Yaskawa INFORM job: X2_34(P)(-165,-90).JBI

/JOB
//NAME X2_34(P)(-165,-90)
//POS
///NPOS 175,175,175,10,0,0
///TOOL 0
///POSTYPE PULSE
///PULSE
C00000=39612,-76551,-106625,-19964,71626,-76894
C00001=136747,-74177,-105509,-19364,71994,-77223
C00002=161484,-91945,-110261,-14957,103238,-71453
C00003=108557,-106327,-63424,-3944,69973,-81240
C00004=108101,-105157,-58666,-3986,67629,-81319
C00005=107910,-104606,-56713,-4004,66704,-81354
C00006=107850,-103240,-54402,-4023,65983,-81349
C00007=107869,-103453,-54807,-4020,66123,-81348
C00008=107897,-103507,-54813,-4022,66100,-81337
C00009=107488,-105602,-55530,-4025,65447,-81456
C00010=107897,-103507,-54813,-4022,66100,-81337
C00011=108089,-104086,-56785,-4002,67023,-81302
C00012=108547,-105331,-61592,-3959,69358,-81223
C00013=104324,-140520,-91585,-2551,64945,-84379
C00014=108507,-122565,-87623,-3050,71648,-81402
C00015=108151,-121446,-83013,-3052,69376,-81469
C00016=108261,-118225,-79182,-3077,68679,-81414
C00017=108248,-117713,-78438,-3081,68485,-81412
C00018=107960,-119858,-79317,-3061,67913,-81499
C00019=108018,-119853,-79323,-3067,67922,-81479
C00020=107613,-122457,-80135,-3040,67069,-81600
C00021=108018,-119853,-79323,-3067,67922,-81479
C00022=108166,-120422,-81226,-3065,68804,-81449
C00023=108523,-121621,-85875,-3062,71060,-81382
C00024=103983,-152784,-104117,29,47198,-80645
C00025=107925,-135086,-100462,-1830,53864,-79007
C00026=108009,-130425,-94870,-1890,52821,-78954
C00027=108095,-127409,-91509,-1942,52305,-78908
C00028=108095,-126631,-90337,-1950,51984,-78902
C00029=107997,-127624,-90886,-1911,51808,-78940
C00030=108092,-127668,-90899,-1953,51796,-78900
C00031=107688,-130656,-91794,-1800,50803,-79052
C00032=108092,-127668,-90899,-1953,51796,-78900
C00033=108059,-129495,-93147,-1927,52240,-78922
C00034=107976,-134157,-98754,-1865,53292,-78976
C00035=177778,-171467,-115875,-22983,53224,-57909
C00036=173225,-131569,-103985,-1828,82945,-64027
C00037=174834,-131579,-99933,-1874,80485,-63443
C00038=175501,-131430,-98256,-1893,79546,-63202
C00039=175652,-130307,-96214,-1900,78870,-63140
C00040=175501,-131430,-98256,-1893,79546,-63202
C00041=175673,-130387,-96489,-1900,78999,-63135
C00042=177249,-132864,-97254,-1939,78235,-62586
C00043=175673,-130387,-96489,-1900,78999,-63135
C00044=175002,-130579,-98183,-1880,79926,-63378
C00045=173387,-130693,-102281,-1834,82351,-63963
C00046=183807,-145514,-102399,-23160,59516,-56806
C00047=173742,-122117,-87314,-5245,73809,-63439
C00048=174955,-120554,-82580,-5392,71786,-62928
C00049=175454,-119846,-80647,-5453,70997,-62718
C00050=175604,-118612,-78506,-5486,70327,-62635
C00051=175579,-118770,-78792,-5481,70420,-62648
C00052=175582,-118807,-78841,-5481,70431,-62647
C00053=177158,-120803,-79498,-5617,69918,-62073
C00054=175582,-118807,-78841,-5481,70431,-62647
C00055=175081,-119542,-80788,-5418,71215,-62858
C00056=173863,-121178,-85561,-5269,73223,-63371
C00057=178906,-130545,-89223,-5416,71014,-61548
C00058=173071,-106231,-63228,-1896,70899,-63899
C00059=174678,-104574,-58322,-1958,68769,-63315
C00060=175345,-103832,-56313,-1985,67930,-63072
C00061=175495,-102440,-53993,-1998,67222,-63009
C00062=175462,-102665,-54381,-1995,67344,-63022
C00063=175499,-102701,-54366,-1997,67317,-63009
C00064=177075,-104318,-54954,-2039,66885,-62461
C00065=175499,-102701,-54366,-1997,67317,-63009
C00066=174829,-103469,-56394,-1970,68154,-63253
C00067=173213,-105197,-61348,-1906,70277,-63841
C00068=156325,-82511,-105508,-20476,72304,-69745
C00069=137289,-84891,-120500,-10173,76813,-76449
C00070=137303,-139323,-128947,-10263,31295,-76421
C00071=31263,-162610,-128854,-9653,11963,-76756
C00072=-11604,-169116,-125244,-11553,23484,-75880
C00073=-126218,-114256,-117174,-36511,17097,-65041
C00074=-135014,-119633,-103449,-15272,86576,-49606
C00075=-106915,-105368,-62725,-601,70273,-77124
C00076=-106469,-104199,-57962,-625,67946,-76958
C00077=-106427,-102978,-55809,-630,67247,-76940
C00078=-106243,-102289,-53695,-641,66303,-76872
C00079=-106247,-102493,-54033,-640,66406,-76874
C00080=-106414,-102537,-54077,-634,66410,-76931
C00081=-105966,-104617,-54795,-653,65787,-76773
C00082=-106414,-102537,-54077,-634,66410,-76931
C00083=-106600,-103115,-56051,-624,67326,-77000
C00084=-107042,-104359,-60863,-599,69645,-77164
C00085=-104685,-138629,-91180,-1583,66049,-76219
C00086=-106630,-121517,-86856,-1571,71994,-76952
C00087=-106291,-120404,-82245,-1626,69736,-76803
C00088=-106369,-118603,-80003,-1623,69281,-76825
C00089=-106273,-117758,-77970,-1641,68465,-76779
C00090=-106369,-117325,-78035,-1630,68726,-76817
C00091=-105806,-121493,-79397,-1702,67435,-76600
C00092=-106260,-118916,-78588,-1645,68251,-76772
C00093=-106400,-119484,-80492,-1621,69128,-76833
C00094=-106737,-120682,-85145,-1565,71368,-76981
C00095=-103582,-154725,-104423,-7901,46985,-74327
C00096=-105847,-133932,-99601,-6432,54310,-75790
C00097=-106008,-129334,-94017,-6450,53230,-75789
C00098=-106186,-126781,-91574,-6391,53025,-75850
C00099=-106032,-126404,-89711,-6537,52091,-75726
C00100=-106043,-126517,-89981,-6523,52197,-75738
C00101=-106189,-126587,-90026,-6461,52177,-75798
C00102=-105733,-129532,-90915,-6744,51254,-75544
C00103=-108012,-126988,-90135,-5688,51903,-76547
C00104=-111352,-129424,-92548,-4223,51933,-77951
C00105=-115848,-139750,-99582,-2280,50777,-79810
C00106=-128118,-112747,-93321,3474,64214,-79770
C00107=-127528,-110232,-88265,3324,62374,-79603
C00108=-131543,-95227,-82196,6801,72600,-80548
C00109=-127385,-98872,-82575,10626,69652,-79105
C00110=-128633,-104119,-85497,7673,66573,-79856
C00111=-133482,-114738,-94073,7136,65366,-81719
C00112=-120617,-145215,-100672,6502,46666,-80493
C00113=-128060,-118279,-84808,1730,71284,-79517
C00114=-126715,-104396,-76461,1008,79558,-78921
C00115=-127226,-103966,-73572,1025,78008,-79108
C00116=-114164,-103931,-73405,641,77785,-74653
C00117=-113472,-104261,-76398,617,79454,-74408
C00118=-113406,-115635,-84087,94,73198,-74379
C00119=-120607,-140483,-89927,5432,60853,-78778
C00120=-127870,-111428,-59268,1524,79956,-81377
C00121=-127569,-111674,-55269,1588,77364,-81314
C00122=-128901,-111086,-52825,1362,76187,-81748
C00123=-121722,-111262,-52306,7471,75604,-79134
C00124=-120160,-111882,-54772,7701,76655,-78573
C00125=-121798,-117083,-61165,7391,78047,-79010
C00126=-128072,-118466,-109287,-15603,91940,-64780
C00127=-126218,-114256,-117174,-36511,17097,-65041
C00128=-118793,-153239,-128782,-32477,23422,-65112
C00129=-11604,-169116,-125244,-11553,23484,-75880
C00130=137287,-84892,-120500,-10191,64594,-76446
C00131=160620,-101266,-113002,-23179,68693,-67515
C00132=129742,-123426,-96067,-9724,56983,-77796
C00133=128383,-112088,-89880,-8248,62649,-78796
C00134=128703,-94902,-82763,-7804,73898,-79469
C00135=128761,-94479,-81272,-15441,73939,-79565
C00136=132411,-100510,-85687,-14454,71493,-77985
C00137=121120,-127859,-96593,-6406,52485,-80997
C00138=120597,-141128,-100343,-6158,49851,-81075
C00139=130265,-122623,-86303,-8823,68773,-76108
C00140=128227,-104700,-77042,-7266,80096,-77610
C00141=128783,-104516,-74147,-7313,78472,-77326
C00142=116886,-104728,-74108,-6967,77291,-81346
C00143=115094,-104918,-77164,-6860,78909,-82052
C00144=115427,-113226,-83932,-6693,75026,-81747
C00145=120594,-141153,-90526,-5480,61036,-81662
C00146=128321,-87817,-54145,-10439,89447,-79015
C00147=127523,-89347,-51051,-10580,86699,-79052
C00148=128055,-89411,-48930,-10495,85448,-78769
C00149=116170,-89524,-49026,-12471,83824,-82572
C00150=114624,-89429,-51130,-12692,84904,-83201
C00151=116009,-88102,-54303,-12461,87687,-83015
C00152=137164,-110674,-71119,11845,85280,-74888
C00153=151370,-92876,-56112,13362,82896,-70290
C00154=153915,-93323,-52552,13704,80129,-69731
C00155=156453,-92356,-50350,13999,78877,-69014
C00156=166960,-85922,-47968,14858,78858,-65431
C00157=165279,-86575,-50027,14687,80058,-65864
C00158=162548,-86326,-53594,14393,82787,-66479
C00159=168553,-109199,-82190,2412,78268,-65016
C00160=153192,-88821,-70941,3038,99890,-61607
C00161=155008,-91116,-68349,3347,97048,-61054
C00162=157187,-90450,-66010,3737,95856,-60347
C00163=166145,-83282,-63279,5372,97344,-57219
C00164=164891,-83194,-65061,5170,98565,-57601
C00165=162880,-81038,-67608,4859,101356,-58186
C00166=167198,-112039,-93522,-10714,66136,-64798
C00167=163968,-83154,-82219,2627,109012,-67999
C00168=165195,-87569,-80699,2798,105770,-67633
C00169=166313,-88762,-79160,2976,104173,-67275
C00170=157667,-97229,-82374,1388,102036,-70348
C00171=155365,-96855,-84468,975,103550,-71144
C00172=154440,-92394,-86138,821,106880,-71447
C00173=136747,-74177,-105509,-19364,71994,-77223
C00174=39612,-76551,-106625,-19964,71626,-76894
BC00000=295309,515546,1075139
BC00001=353519,294132,1075139
BC00002=353519,214242,1075139
BC00003=342438,159660,1075139
BC00004=342438,159660,1075139
BC00005=342438,159660,1075139
BC00006=342438,159660,1075139
BC00007=342438,159660,1075139
BC00008=342438,159660,1075139
BC00009=342438,159660,1075139
BC00010=342438,159660,1075139
BC00011=342438,159660,1075139
BC00012=342438,159660,1075139
BC00013=342356,136521,1075139
BC00014=342356,136521,1075139
BC00015=342356,136521,1075139
BC00016=342356,136521,1075139
BC00017=342356,136521,1075139
BC00018=342356,136521,1075139
BC00019=342356,136521,1075139
BC00020=342356,136521,1075139
BC00021=342356,136521,1075139
BC00022=342356,136521,1075139
BC00023=342356,136521,1075139
BC00024=339297,143778,1075139
BC00025=339297,143778,1075139
BC00026=339297,143778,1075139
BC00027=339297,143778,1075139
BC00028=339297,143778,1075139
BC00029=339297,143778,1075139
BC00030=339297,143778,1075139
BC00031=339297,143778,1075139
BC00032=339297,143778,1075139
BC00033=339297,143778,1075139
BC00034=339297,143778,1075139
BC00035=316428,128559,1075139
BC00036=316320,82093,1075139
BC00037=316320,82093,1075139
BC00038=316320,82093,1075139
BC00039=316320,82093,1075139
BC00040=316320,82093,1075139
BC00041=316320,82093,1075139
BC00042=316320,82093,1075139
BC00043=316320,82093,1075139
BC00044=316320,82093,1075139
BC00045=316320,82093,1075139
BC00046=316428,128559,1075139
BC00047=316362,120660,1075139
BC00048=316362,120660,1075139
BC00049=316362,120660,1075139
BC00050=316362,120660,1075139
BC00051=316362,120660,1075139
BC00052=316362,120660,1075139
BC00053=316362,120660,1075139
BC00054=316362,120660,1075139
BC00055=316362,120660,1075139
BC00056=316362,120660,1075139
BC00057=316362,120660,1075139
BC00058=316494,143798,1075139
BC00059=316494,143798,1075139
BC00060=316494,143798,1075139
BC00061=316494,143798,1075139
BC00062=316494,143798,1075139
BC00063=316494,143798,1075139
BC00064=316494,143798,1075139
BC00065=316494,143798,1075139
BC00066=316494,143798,1075139
BC00067=316494,143798,1075139
BC00068=381880,223521,1075139
BC00069=353800,266120,1075139
BC00070=353800,266120,1075139
BC00071=379757,63718,1075139
BC00072=335939,159824,1075139
BC00073=312616,52052,1075139
BC00074=340737,74809,1075139
BC00075=348041,96035,1075139
BC00076=348041,96035,1075139
BC00077=348041,96035,1075139
BC00078=348041,96035,1075139
BC00079=348041,96035,1075139
BC00080=348041,96035,1075139
BC00081=348041,96035,1075139
BC00082=348041,96035,1075139
BC00083=348041,96035,1075139
BC00084=348041,96035,1075139
BC00085=347852,119343,1075139
BC00086=347852,119343,1075139
BC00087=347852,119343,1075139
BC00088=347852,119343,1075139
BC00089=347852,119343,1075139
BC00090=347852,119343,1075139
BC00091=347852,119343,1075139
BC00092=347852,119343,1075139
BC00093=347852,119343,1075139
BC00094=347852,119343,1075139
BC00095=347961,111500,1075139
BC00096=347961,111500,1075139
BC00097=347961,111500,1075139
BC00098=347961,111500,1075139
BC00099=347961,111500,1075139
BC00100=347961,111500,1075139
BC00101=347961,111500,1075139
BC00102=347961,111500,1075139
BC00103=347961,111500,1075139
BC00104=347961,111500,1075139
BC00105=347961,111500,1075139
BC00106=359170,99356,1075139
BC00107=359170,99356,1075139
BC00108=359170,99356,1075139
BC00109=359170,99356,1075139
BC00110=359169,99356,1075136
BC00111=359170,99356,1075138
BC00112=343018,99541,1075139
BC00113=358041,112918,1075139
BC00114=358041,112918,1075139
BC00115=358041,112918,1075139
BC00116=358041,112918,1075139
BC00117=358041,112918,1075139
BC00118=358041,112918,1075139
BC00119=343061,115981,1075139
BC00120=353714,134453,1075139
BC00121=353714,134453,1075139
BC00122=353714,134453,1075139
BC00123=353714,134453,1075139
BC00124=353714,134453,1075139
BC00125=353714,134453,1075139
BC00126=340737,74809,1075139
BC00127=312616,52052,1075139
BC00128=312616,52052,1075139
BC00129=335939,159824,1075139
BC00130=353801,266119,1075139
BC00131=381880,223521,1075139
BC00132=352343,156430,1075139
BC00133=352343,156430,1075139
BC00134=352343,156430,1075139
BC00135=352343,156430,1075139
BC00136=352343,156430,1075139
BC00137=352343,156430,1075139
BC00138=343465,156897,1075139
BC00139=349372,143881,1075139
BC00140=349372,143881,1075139
BC00141=349372,143881,1075139
BC00142=349372,143881,1075139
BC00143=349372,143881,1075139
BC00144=349372,143881,1075139
BC00145=343515,140305,1075139
BC00146=339496,150749,1057604
BC00147=339496,150749,1057604
BC00148=339496,150749,1057604
BC00149=339496,150749,1057604
BC00150=339496,150749,1057604
BC00151=339496,150749,1057604
BC00152=341295,130990,1075139
BC00153=330397,138794,1057889
BC00154=330397,138794,1057889
BC00155=330397,138794,1057889
BC00156=330397,138794,1057889
BC00157=330397,138794,1057889
BC00158=330397,138794,1057889
BC00159=337522,139852,1075139
BC00160=315665,114809,1075139
BC00161=315665,114809,1075139
BC00162=315665,114809,1075139
BC00163=315665,114809,1075139
BC00164=315665,114809,1075139
BC00165=315665,114809,1075139
BC00166=337528,156420,1075139
BC00167=308596,87959,1075139
BC00168=308596,87959,1075139
BC00169=308596,87959,1075139
BC00170=308596,87959,1075139
BC00171=308596,87959,1075139
BC00172=308596,87959,1075139
BC00173=353519,294132,1075139
BC00174=295309,515546,1075139
EC00000=1463287,372643
EC00001=1463287,372643
EC00002=1463287,372643
EC00003=1463287,372643
EC00004=1463287,372643
EC00005=1463287,372643
EC00006=1463287,372643
EC00007=1463287,372643
EC00008=1463287,372643
EC00009=1463287,372643
EC00010=1463287,372643
EC00011=1463287,372643
EC00012=1463287,372643
EC00013=1463287,372643
EC00014=1463287,372643
EC00015=1463287,372643
EC00016=1463287,372643
EC00017=1463287,372643
EC00018=1463287,372643
EC00019=1463287,372643
EC00020=1463287,372643
EC00021=1463287,372643
EC00022=1463287,372643
EC00023=1463287,372643
EC00024=1463287,372643
EC00025=1463287,372643
EC00026=1463287,372643
EC00027=1463287,372643
EC00028=1463287,372643
EC00029=1463287,372643
EC00030=1463287,372643
EC00031=1463287,372643
EC00032=1463287,372643
EC00033=1463287,372643
EC00034=1463287,372643
EC00035=1463287,372643
EC00036=1463287,372643
EC00037=1463287,372643
EC00038=1463287,372643
EC00039=1463287,372643
EC00040=1463287,372643
EC00041=1463287,372643
EC00042=1463287,372643
EC00043=1463287,372643
EC00044=1463287,372643
EC00045=1463287,372643
EC00046=1463287,372643
EC00047=1463287,372643
EC00048=1463287,372643
EC00049=1463287,372643
EC00050=1463287,372643
EC00051=1463287,372643
EC00052=1463287,372643
EC00053=1463287,372643
EC00054=1463287,372643
EC00055=1463287,372643
EC00056=1463287,372643
EC00057=1463287,372643
EC00058=1463287,372643
EC00059=1463287,372643
EC00060=1463287,372643
EC00061=1463287,372643
EC00062=1463287,372643
EC00063=1463287,372643
EC00064=1463287,372643
EC00065=1463287,372643
EC00066=1463287,372643
EC00067=1463287,372643
EC00068=1463287,372643
EC00069=1463287,372643
EC00070=1463287,372643
EC00071=1463287,372643
EC00072=1595090,-179995
EC00073=1729339,-740307
EC00074=1729339,-740307
EC00075=1729339,-740307
EC00076=1729339,-740307
EC00077=1729339,-740307
EC00078=1729339,-740307
EC00079=1729339,-740307
EC00080=1729339,-740307
EC00081=1729339,-740307
EC00082=1729339,-740307
EC00083=1729339,-740307
EC00084=1729339,-740307
EC00085=1729339,-740307
EC00086=1729339,-740307
EC00087=1729339,-740307
EC00088=1729339,-740307
EC00089=1729339,-740307
EC00090=1729339,-740307
EC00091=1729339,-740307
EC00092=1729339,-740307
EC00093=1729339,-740307
EC00094=1729339,-740307
EC00095=1729339,-740307
EC00096=1729339,-740307
EC00097=1729339,-740307
EC00098=1729339,-740307
EC00099=1729339,-740307
EC00100=1729339,-740307
EC00101=1729339,-740307
EC00102=1729339,-740307
EC00103=1729339,-740307
EC00104=1729339,-740307
EC00105=1729339,-740307
EC00106=1729339,-740307
EC00107=1729339,-740307
EC00108=1729339,-740307
EC00109=1729339,-740307
EC00110=1729341,-740306
EC00111=1729340,-740307
EC00112=1729339,-740307
EC00113=1729339,-740307
EC00114=1729339,-740307
EC00115=1729339,-740307
EC00116=1729339,-740307
EC00117=1729339,-740307
EC00118=1729339,-740307
EC00119=1729339,-740307
EC00120=1729339,-740307
EC00121=1729339,-740307
EC00122=1729339,-740307
EC00123=1729339,-740307
EC00124=1729339,-740307
EC00125=1729339,-740307
EC00126=1729339,-740307
EC00127=1729339,-740307
EC00128=1729339,-740307
EC00129=1595090,-179995
EC00130=1463287,372643
EC00131=1463287,372643
EC00132=1463287,372643
EC00133=1463287,372643
EC00134=1463287,372643
EC00135=1463287,372643
EC00136=1463287,372643
EC00137=1463287,372643
EC00138=1463287,372643
EC00139=1463287,372643
EC00140=1463287,372643
EC00141=1463287,372643
EC00142=1463287,372643
EC00143=1463287,372643
EC00144=1463287,372643
EC00145=1463287,372643
EC00146=1463287,372643
EC00147=1463287,372643
EC00148=1463287,372643
EC00149=1463287,372643
EC00150=1463287,372643
EC00151=1463287,372643
EC00152=1463287,372643
EC00153=1463287,372643
EC00154=1463287,372643
EC00155=1463287,372643
EC00156=1463287,372643
EC00157=1463287,372643
EC00158=1463287,372643
EC00159=1463287,372643
EC00160=1463287,372643
EC00161=1463287,372643
EC00162=1463287,372643
EC00163=1463287,372643
EC00164=1463287,372643
EC00165=1463287,372643
EC00166=1463287,372643
EC00167=1463287,372643
EC00168=1463287,372643
EC00169=1463287,372643
EC00170=1463287,372643
EC00171=1463287,372643
EC00172=1463287,372643
EC00173=1463287,372643
EC00174=1463287,372643
///POSTYPE BASE
///RECTAN
///RCONF 0,0,0,0,1,0,0,0,0,0,0,0,0,0,0,0,0,0,0,0,0,0,0,0
P00006=2.006,1.622,-0.565,0.0000,0.0000,0.0000
P00021=0.073,2.058,-0.109,0.0000,0.0000,0.0000
P00022=2.006,1.622,-0.565,0.0000,0.0000,0.0000
///RCONF 0,0,0,0,0,0,0,0,0,0,0,0,0,0,0,0,0,0,0,0,0,0,0,0
P00023=-2.957,-4.083,2.762,0.0000,0.0000,0.0000
P00024=-1.466,-0.226,-0.419,0.0000,0.0000,0.0000
P00025=3.643,0.007,-2.585,0.0000,0.0000,0.0000
P00026=2.644,0.055,-2.583,0.0000,0.0000,0.0000
///RCONF 0,0,0,0,1,0,0,0,0,0,0,0,0,0,0,0,0,0,0,0,0,0,0,0
P00034=-8.151,9.743,-4.393,0.0000,0.0000,0.0000
///RCONF 0,0,0,0,0,0,0,0,0,0,0,0,0,0,0,0,0,0,0,0,0,0,0,0
P00035=0.390,-0.027,1.040,0.0000,0.0000,0.0000
P00036=-2.434,0.084,0.197,0.0000,0.0000,0.0000
//INST
///DATE 2024/12/04 09:57
///ATTR SC,RW
///GROUP1 RB1,BS1
///GROUP2 ST1
NOP
'X2_34(P)(-165,-90)
MOVJ C00000 BC00000 VJ=100.00  +MOVJ EC00000 VJ=100.00
MOVJ C00001 BC00001 VJ=100.00  +MOVJ EC00001 VJ=100.00
MOVJ C00002 BC00002 VJ=100.00  +MOVJ EC00002 VJ=100.00
'Path S3213
SFTOF3D
MOVJ C00003 BC00003 VJ=100.00  +MOVJ EC00003 VJ=100.00
MOVL C00004 BC00004 V=800.0  +MOVJ EC00004 VJ=100.00
SMOVL C00005 BC00005 V=166.7  +MOVJ EC00005
SREFP 3 C00006 BC00006  +REFP EC00006
CALL JOB:SEARCH-R1-S13D
SET P021 P006
SFTON3D P021
SMOVL C00007 BC00007 V=166.7  +MOVJ EC00007
SMOVL C00008 BC00008 V=166.7  +MOVJ EC00008
SREFP 3 C00009 BC00009  +REFP EC00009
CALL JOB:SEARCH-R1-S13D
SET P021 P006
SFTON3D P021
SMOVL C00010 BC00010 V=166.7  +MOVJ EC00010
MOVL C00011 BC00011 V=800.0  +MOVJ EC00011 VJ=100.00
MOVL C00012 BC00012 V=1000.0  +MOVJ EC00012 VJ=100.00
'EndPath S3213
MOVJ C00013 BC00013 VJ=100.00  +MOVJ EC00013 VJ=100.00
'Path S3214
SFTOF3D
MOVJ C00014 BC00014 VJ=100.00  +MOVJ EC00014 VJ=100.00
MOVL C00015 BC00015 V=800.0  +MOVJ EC00015 VJ=100.00
SMOVL C00016 BC00016 V=166.7  +MOVJ EC00016
SREFP 3 C00017 BC00017  +REFP EC00017
CALL JOB:SEARCH-R1-S13D
SET P022 P006
SFTON3D P022
SMOVL C00018 BC00018 V=166.7  +MOVJ EC00018
SMOVL C00019 BC00019 V=166.7  +MOVJ EC00019
SREFP 3 C00020 BC00020  +REFP EC00020
CALL JOB:SEARCH-R1-S13D
SET P022 P006
SFTON3D P022
SMOVL C00021 BC00021 V=166.7  +MOVJ EC00021
MOVL C00022 BC00022 V=800.0  +MOVJ EC00022 VJ=100.00
MOVL C00023 BC00023 V=1000.0  +MOVJ EC00023 VJ=100.00
'EndPath S3214
MOVJ C00024 BC00024 VJ=100.00  +MOVJ EC00024 VJ=100.00
'Path S3215
SFTOF3D
MOVJ C00025 BC00025 VJ=100.00  +MOVJ EC00025 VJ=100.00
MOVL C00026 BC00026 V=800.0  +MOVJ EC00026 VJ=100.00
SMOVL C00027 BC00027 V=166.7  +MOVJ EC00027
SREFP 3 C00028 BC00028  +REFP EC00028
CALL JOB:SEARCH-R1-S13D
SET P023 P006
SFTON3D P023
SMOVL C00029 BC00029 V=166.7  +MOVJ EC00029
SMOVL C00030 BC00030 V=166.7  +MOVJ EC00030
SREFP 3 C00031 BC00031  +REFP EC00031
CALL JOB:SEARCH-R1-S13D
SET P023 P006
SFTON3D P023
SMOVL C00032 BC00032 V=166.7  +MOVJ EC00032
MOVL C00033 BC00033 V=800.0  +MOVJ EC00033 VJ=100.00
MOVL C00034 BC00034 V=1000.0  +MOVJ EC00034 VJ=100.00
'EndPath S3215
MOVJ C00035 BC00035 VJ=100.00  +MOVJ EC00035 VJ=100.00
'Path S3216
SFTOF3D
MOVJ C00036 BC00036 VJ=100.00  +MOVJ EC00036 VJ=100.00
MOVL C00037 BC00037 V=800.0  +MOVJ EC00037 VJ=100.00
SMOVL C00038 BC00038 V=166.7  +MOVJ EC00038
SREFP 3 C00039 BC00039  +REFP EC00039
CALL JOB:SEARCH-R1-S13D
SET P024 P006
SFTON3D P024
SMOVL C00040 BC00040 V=166.7  +MOVJ EC00040
SMOVL C00041 BC00041 V=166.7  +MOVJ EC00041
SREFP 3 C00042 BC00042  +REFP EC00042
CALL JOB:SEARCH-R1-S13D
SET P024 P006
SFTON3D P024
SMOVL C00043 BC00043 V=166.7  +MOVJ EC00043
MOVL C00044 BC00044 V=800.0  +MOVJ EC00044 VJ=100.00
MOVL C00045 BC00045 V=1000.0  +MOVJ EC00045 VJ=100.00
'EndPath S3216
MOVJ C00046 BC00046 VJ=100.00  +MOVJ EC00046 VJ=100.00
'Path S3217
SFTOF3D
MOVJ C00047 BC00047 VJ=100.00  +MOVJ EC00047 VJ=100.00
MOVL C00048 BC00048 V=800.0  +MOVJ EC00048 VJ=100.00
SMOVL C00049 BC00049 V=166.7  +MOVJ EC00049
SREFP 3 C00050 BC00050  +REFP EC00050
CALL JOB:SEARCH-R1-S13D
SET P025 P006
SFTON3D P025
SMOVL C00051 BC00051 V=166.7  +MOVJ EC00051
SMOVL C00052 BC00052 V=166.7  +MOVJ EC00052
SREFP 3 C00053 BC00053  +REFP EC00053
CALL JOB:SEARCH-R1-S13D
SET P025 P006
SFTON3D P025
SMOVL C00054 BC00054 V=166.7  +MOVJ EC00054
MOVL C00055 BC00055 V=800.0  +MOVJ EC00055 VJ=100.00
MOVL C00056 BC00056 V=1000.0  +MOVJ EC00056 VJ=100.00
'EndPath S3217
MOVJ C00057 BC00057 VJ=100.00  +MOVJ EC00057 VJ=100.00
'Path S3218
SFTOF3D
MOVJ C00058 BC00058 VJ=100.00  +MOVJ EC00058 VJ=100.00
MOVL C00059 BC00059 V=800.0  +MOVJ EC00059 VJ=100.00
SMOVL C00060 BC00060 V=166.7  +MOVJ EC00060
SREFP 3 C00061 BC00061  +REFP EC00061
CALL JOB:SEARCH-R1-S13D
SET P026 P006
SFTON3D P026
SMOVL C00062 BC00062 V=166.7  +MOVJ EC00062
SMOVL C00063 BC00063 V=166.7  +MOVJ EC00063
SREFP 3 C00064 BC00064  +REFP EC00064
CALL JOB:SEARCH-R1-S13D
SET P026 P006
SFTON3D P026
SMOVL C00065 BC00065 V=166.7  +MOVJ EC00065
MOVL C00066 BC00066 V=800.0  +MOVJ EC00066 VJ=100.00
MOVL C00067 BC00067 V=1000.0  +MOVJ EC00067 VJ=100.00
'EndPath S3218
'obrot
MOVJ C00068 BC00068 VJ=100.00  +MOVJ EC00068 VJ=100.00
MOVJ C00069 BC00069 VJ=100.00  +MOVJ EC00069 VJ=100.00
MOVJ C00070 BC00070 VJ=100.00  +MOVJ EC00070 VJ=100.00
MOVJ C00071 BC00071 VJ=100.00  +MOVJ EC00071 VJ=100.00
MOVJ C00072 BC00072 VJ=100.00  +MOVJ EC00072 VJ=100.00
MOVJ C00073 BC00073 VJ=100.00  +MOVJ EC00073 VJ=100.00
MOVJ C00074 BC00074 VJ=100.00  +MOVJ EC00074 VJ=100.00
'
'Path S3219
SFTOF3D
MOVJ C00075 BC00075 VJ=100.00  +MOVJ EC00075 VJ=100.00
MOVL C00076 BC00076 V=800.0  +MOVJ EC00076 VJ=100.00
SMOVL C00077 BC00077 V=166.7  +MOVJ EC00077
SREFP 3 C00078 BC00078  +REFP EC00078
CALL JOB:SEARCH-R1-S13D
SET P034 P006
SFTON3D P034
SMOVL C00079 BC00079 V=166.7  +MOVJ EC00079
SMOVL C00080 BC00080 V=166.7  +MOVJ EC00080
SREFP 3 C00081 BC00081  +REFP EC00081
CALL JOB:SEARCH-R1-S13D
SET P034 P006
SFTON3D P034
SMOVL C00082 BC00082 V=166.7  +MOVJ EC00082
MOVL C00083 BC00083 V=800.0  +MOVJ EC00083 VJ=100.00
MOVL C00084 BC00084 V=1000.0  +MOVJ EC00084 VJ=100.00
'EndPath S3219
MOVJ C00085 BC00085 VJ=100.00  +MOVJ EC00085 VJ=100.00
'Path S3220
SFTOF3D
MOVJ C00086 BC00086 VJ=100.00  +MOVJ EC00086 VJ=100.00
MOVL C00087 BC00087 V=800.0  +MOVJ EC00087 VJ=100.00
SMOVL C00088 BC00088 V=166.7  +MOVJ EC00088
SREFP 3 C00089 BC00089  +REFP EC00089
CALL JOB:SEARCH-R1-S13D
SET P035 P006
SFTON3D P035
SMOVL C00090 BC00090 V=166.7  +MOVJ EC00090
SREFP 3 C00091 BC00091  +REFP EC00091
CALL JOB:SEARCH-R1-S13D
SET P035 P006
SFTON3D P035
SMOVL C00092 BC00092 V=166.7  +MOVJ EC00092
MOVL C00093 BC00093 V=800.0  +MOVJ EC00093 VJ=100.00
MOVL C00094 BC00094 V=1000.0  +MOVJ EC00094 VJ=100.00
'EndPath S3220
MOVJ C00095 BC00095 VJ=100.00  +MOVJ EC00095 VJ=100.00
'Path S3221
SFTOF3D
MOVJ C00096 BC00096 VJ=100.00  +MOVJ EC00096 VJ=100.00
MOVL C00097 BC00097 V=800.0  +MOVJ EC00097 VJ=100.00
SMOVL C00098 BC00098 V=166.7  +MOVJ EC00098
SREFP 3 C00099 BC00099  +REFP EC00099
CALL JOB:SEARCH-R1-S13D
SET P036 P006
SFTON3D P036
SMOVL C00100 BC00100 V=166.7  +MOVJ EC00100
SMOVL C00101 BC00101 V=166.7  +MOVJ EC00101
SREFP 3 C00102 BC00102  +REFP EC00102
CALL JOB:SEARCH-R1-S13D
SET P036 P006
SFTON3D P036
SMOVL C00103 BC00103 V=166.7  +MOVJ EC00103
MOVL C00104 BC00104 V=800.0  +MOVJ EC00104 VJ=100.00
MOVL C00105 BC00105 V=1000.0  +MOVJ EC00105 VJ=100.00
'EndPath S3221
'Path W3222
SFTOF3D
SFTON3D P036
MOVJ C00106 BC00106 VJ=100.00  +MOVJ EC00106 VJ=100.00
SMOVL C00107 BC00107 V=800.0  +MOVJ EC00107
MACRO1 MJ#(0) ARGF21
SMOVL C00108 BC00108 V=166.7 PL=0  +MOVJ EC00108
ARCON
SMOVL C00109 BC00109 V=11.7  +MOVJ EC00109
ARCOF
SMOVL C00110 BC00110 V=800.0  +MOVJ EC00110
SMOVL C00111 BC00111 V=1000.0  +MOVJ EC00111
SFTOF3D
'EndPath W3222
MOVJ C00112 BC00112 VJ=100.00  +MOVJ EC00112 VJ=100.00
'Path W3223
SFTOF3D
SFTON3D P035
MOVJ C00113 BC00113 VJ=100.00  +MOVJ EC00113 VJ=100.00
SMOVL C00114 BC00114 V=800.0  +MOVJ EC00114
SMOVL C00115 BC00115 V=166.7 PL=0  +MOVJ EC00115
ARCON
SMOVL C00116 BC00116 V=11.7  +MOVJ EC00116
ARCOF
SMOVL C00117 BC00117 V=800.0  +MOVJ EC00117
SMOVL C00118 BC00118 V=1000.0  +MOVJ EC00118
SFTOF3D
'EndPath W3223
MOVJ C00119 BC00119 VJ=100.00  +MOVJ EC00119 VJ=100.00
'Path W3224
SFTOF3D
SFTON3D P034
MOVJ C00120 BC00120 VJ=100.00  +MOVJ EC00120 VJ=100.00
SMOVL C00121 BC00121 V=800.0  +MOVJ EC00121
SMOVL C00122 BC00122 V=166.7 PL=0  +MOVJ EC00122
ARCON
SMOVL C00123 BC00123 V=11.7  +MOVJ EC00123
ARCOF
SMOVL C00124 BC00124 V=800.0  +MOVJ EC00124
SMOVL C00125 BC00125 V=1000.0  +MOVJ EC00125
SFTOF3D
'EndPath W3224
'obrot
MOVJ C00126 BC00126 VJ=100.00  +MOVJ EC00126 VJ=100.00
MOVJ C00127 BC00127 VJ=100.00  +MOVJ EC00127 VJ=100.00
MOVJ C00128 BC00128 VJ=100.00  +MOVJ EC00128 VJ=100.00
MOVJ C00129 BC00129 VJ=100.00  +MOVJ EC00129 VJ=100.00
MOVJ C00130 BC00130 VJ=100.00  +MOVJ EC00130 VJ=100.00
MOVJ C00131 BC00131 VJ=100.00  +MOVJ EC00131 VJ=100.00
'
'Path W3225
SFTOF3D
SFTON3D P023
MOVJ C00132 BC00132 VJ=100.00  +MOVJ EC00132 VJ=100.00
SMOVL C00133 BC00133 V=800.0  +MOVJ EC00133
SMOVL C00134 BC00134 V=166.7 PL=0  +MOVJ EC00134
ARCON
SMOVL C00135 BC00135 V=11.7  +MOVJ EC00135
ARCOF
SMOVL C00136 BC00136 V=800.0  +MOVJ EC00136
SMOVL C00137 BC00137 V=1000.0  +MOVJ EC00137
SFTOF3D
'EndPath W3225
MOVJ C00138 BC00138 VJ=100.00  +MOVJ EC00138 VJ=100.00
'Path W3226
SFTOF3D
SFTON3D P022
MOVJ C00139 BC00139 VJ=100.00  +MOVJ EC00139 VJ=100.00
SMOVL C00140 BC00140 V=800.0  +MOVJ EC00140
SMOVL C00141 BC00141 V=166.7 PL=0  +MOVJ EC00141
ARCON
SMOVL C00142 BC00142 V=11.7  +MOVJ EC00142
ARCOF
SMOVL C00143 BC00143 V=800.0  +MOVJ EC00143
SMOVL C00144 BC00144 V=1000.0  +MOVJ EC00144
SFTOF3D
'EndPath W3226
MOVJ C00145 BC00145 VJ=100.00  +MOVJ EC00145 VJ=100.00
'Path W3227
SFTOF3D
SFTON3D P021
MOVJ C00146 BC00146 VJ=100.00  +MOVJ EC00146 VJ=100.00
SMOVL C00147 BC00147 V=800.0  +MOVJ EC00147
SMOVL C00148 BC00148 V=166.7 PL=0  +MOVJ EC00148
ARCON
SMOVL C00149 BC00149 V=11.7  +MOVJ EC00149
ARCOF
SMOVL C00150 BC00150 V=800.0  +MOVJ EC00150
SMOVL C00151 BC00151 V=1000.0  +MOVJ EC00151
SFTOF3D
'EndPath W3227
MOVJ C00152 BC00152 VJ=100.00  +MOVJ EC00152 VJ=100.00
'Path W3228
SFTOF3D
SFTON3D P026
MOVJ C00153 BC00153 VJ=100.00  +MOVJ EC00153 VJ=100.00
SMOVL C00154 BC00154 V=800.0  +MOVJ EC00154
SMOVL C00155 BC00155 V=166.7 PL=0  +MOVJ EC00155
ARCON
SMOVL C00156 BC00156 V=11.7  +MOVJ EC00156
ARCOF
SMOVL C00157 BC00157 V=800.0  +MOVJ EC00157
SMOVL C00158 BC00158 V=1000.0  +MOVJ EC00158
SFTOF3D
'EndPath W3228
MOVJ C00159 BC00159 VJ=100.00  +MOVJ EC00159 VJ=100.00
'Path W3229
SFTOF3D
SFTON3D P025
MOVJ C00160 BC00160 VJ=100.00  +MOVJ EC00160 VJ=100.00
SMOVL C00161 BC00161 V=800.0  +MOVJ EC00161
SMOVL C00162 BC00162 V=166.7 PL=0  +MOVJ EC00162
ARCON
SMOVL C00163 BC00163 V=11.7  +MOVJ EC00163
ARCOF
SMOVL C00164 BC00164 V=800.0  +MOVJ EC00164
SMOVL C00165 BC00165 V=1000.0  +MOVJ EC00165
SFTOF3D
'EndPath W3229
MOVJ C00166 BC00166 VJ=100.00  +MOVJ EC00166 VJ=100.00
'Path W3230
SFTOF3D
SFTON3D P024
MOVJ C00167 BC00167 VJ=100.00  +MOVJ EC00167 VJ=100.00
SMOVL C00168 BC00168 V=800.0  +MOVJ EC00168
SMOVL C00169 BC00169 V=166.7 PL=0  +MOVJ EC00169
ARCON
SMOVL C00170 BC00170 V=11.7  +MOVJ EC00170
ARCOF
SMOVL C00171 BC00171 V=800.0  +MOVJ EC00171
SMOVL C00172 BC00172 V=1000.0  +MOVJ EC00172
SFTOF3D
'EndPath W3230
MOVJ C00173 BC00173 VJ=100.00  +MOVJ EC00173 VJ=100.00
MOVJ C00174 BC00174 VJ=100.00  +MOVJ EC00174 VJ=100.00
END
